PROGRAM PRG_KFE_RIX_VAC_FS
VAR
END_VAR

//Fast Shutter Valve

fb_TV1K2_VFS_1(
    i_xVeto_Enable:=True,
	i_xPMPS_OK:= TRUE, 
	i_xExt_OK:= TRUE, 
	i_sDevName:= 'TV1K2:VFS:1',	 
	io_fbFFHWO:= g_FastFaultOutput2
);
(*FastFaultOuput*)	
g_FastFaultOutput2.Execute(bAutoReset:= TRUE);

END_PROGRAM

(* stored: Version 1.1.0.1, ProductVersion 3.1.4022.18
   POU PRG_KFE_RIX_VAC_FS: Id {4a8c2d36-37b0-4436-8b46-6263bf0245fa}, SpecialFunc None *)
